(* IEC 61131-3 sources: MessageBox/src/Ar/MessageBox, 3 files *)

(* ---- MessageBox.typ ---- *)
(*
* File: MessageBox.typ
* Copyright (c) 2023 Loupe
* https://loupe.team
*
* This file is part of MessageBox, licensed under the MIT License.
*
*)
(*Popup HMI Control*)

TYPE
	MessageBox_HMI_typ : 	STRUCT
		Layer : MessageBox_Layer_typ;
		TextSnippets : MessageBox_TextSnippets;
		Prompt : HMI_TextBox_typ;
		UserInput : HMI_TextBox_typ;
		Buttons1 : HMI_Button_typ;
		Buttons2 : HMI_Button_typ;
		Buttons3 : HMI_Button_typ;
		Buttons4 : HMI_Button_typ;
		Buttons5 : HMI_Button_typ;
		Internal : MessageBox_HMI_Internal_typ;
	END_STRUCT;
END_TYPE

(*Popup HMI Mapping*)

TYPE
	MessageBox_TextSnippets : 	STRUCT
		Message : STRING[260];
		UserString : STRING[260];
		Buttons1 : STRING[80];
		Buttons2 : STRING[80];
		Buttons3 : STRING[80];
		Buttons4 : STRING[80];
		Buttons5 : STRING[80];
	END_STRUCT;
	MessageBox_Layer_typ : 	STRUCT
		Active : BOOL;
		Status : UINT;
	END_STRUCT;
END_TYPE

(*Structure to create a message*)

TYPE
	MessageBox_Message_typ : 	STRUCT
		Prompt : MessageBox_Message_Prompt_typ;
		Buttons : ARRAY[0..4]OF MessageBox_Button_typ;
		pUserString : UDINT;
		MessageID : UDINT;
	END_STRUCT;
	MessageBox_Message_Prompt_typ : 	STRUCT
		pText : UDINT;
		Index : UINT;
	END_STRUCT;
	MessageBox_Button_typ : 	STRUCT
		pText : UDINT;
		Index : UINT;
		pCmd : UDINT;
	END_STRUCT;
END_TYPE

(*Popup Backend*)

TYPE
	MessageBox_typ : 	STRUCT
		Internal : MessageBox_Internal_typ;
	END_STRUCT;
	MessageBox_Internal_typ : 	STRUCT
		Buffer : Buffer_typ;
	END_STRUCT;
	MessageBox_HMI_Internal_typ : 	STRUCT
		Message : MessageBox_Message_typ;
		_Show : BOOL;
		_CMD : ARRAY[0..4]OF BOOL;
		_ShowEdge : BOOL;
		_ShowDelay : TON;
		_MessageID : UDINT;
	END_STRUCT;
END_TYPE

(*Errors*)

TYPE
	MESSAGE_ERR :
		(
		MESSAGE_ERR_INVALID_ID,
		MESSAGE_ERR_ALREADY_INIT,
		MESSAGE_ERR_OUT_OF_MEMORY,
		MESSAGE_ERR_BUFFER_FULL,
		MESSAGE_ERR_UNINITIALIZED,
		MESSAGE_ERR_EMPTY,
		MESSAGE_ERR_INVALID_POINTER,
		MESSAGE_ERR_
		);
END_TYPE

(* ---- MessageBox.fun ---- *)
(*
* File: MessageBox.fun
* Copyright (c) 2023 Loupe
* https://loupe.team
*
* This file is part of MessageBox, licensed under the MIT License.
*
*)

FUNCTION MessageBox_Init : UDINT (*instantiates a message queue*)
	VAR_INPUT
		QueueSize : USINT;
	END_VAR
END_FUNCTION

FUNCTION MessageBox_AddMsg : UDINT (*adds a normal priority message to the bottom of the list*)
	VAR_INPUT
		Message : UDINT;
		Button1Text : UDINT;
		pCommand1 : UDINT;
		Button2Text : UDINT;
		pCommand2 : UDINT;
	END_VAR
END_FUNCTION

FUNCTION MessageBox_AddMsgTop : UDINT (*adds a high priority message to the top of the list, can bump off the last msg in the buffer*)
	VAR_INPUT
		Message : UDINT;
		Button1Text : UDINT;
		pCommand1 : UDINT;
		Button2Text : UDINT;
		pCommand2 : UDINT;
	END_VAR
END_FUNCTION

FUNCTION PromptBox_AddMsg : UDINT (*adds a normal priority message to the bottom of the list*)
	VAR_INPUT
		Message : UDINT;
		pInputString : UDINT;
		Button1Text : UDINT;
		pCommand1 : UDINT;
		Button2Text : UDINT;
		pCommand2 : UDINT;
	END_VAR
END_FUNCTION

FUNCTION PromptBox_AddMsgTop : UDINT (*adds a high priority message to the top of the list, can bump off the last msg in the buffer*)
	VAR_INPUT
		Message : UDINT;
		pInputString : UDINT;
		Button1Text : UDINT;
		pCommand1 : UDINT;
		Button2Text : UDINT;
		pCommand2 : UDINT;
	END_VAR
END_FUNCTION

FUNCTION MessageBox_RemoveMsg : UDINT (*marks a message for removal based on messageID*)
	VAR_INPUT
		MessageID : UDINT;
	END_VAR
END_FUNCTION

FUNCTION MessageBox_HMI : UDINT (*used to cyclically update messagebox interface with HMI*)
	VAR_INPUT
		MessageBox : MessageBox_HMI_typ;
	END_VAR
END_FUNCTION

FUNCTION MessageBox_Add3BtnMsg : UDINT (*adds a normal priority 3-button message to the bottom of the list*)
	VAR_INPUT
		Message : UDINT;
		Button1Text : UDINT;
		pCommand1 : UDINT;
		Button2Text : UDINT;
		pCommand2 : UDINT;
		Button3Text : UDINT;
		pCommand3 : UDINT;
	END_VAR
END_FUNCTION

FUNCTION MessageBox_Add3BtnMsgTop : UDINT (*adds a high priority 3-button message to the top of the list, can bump off the last msg in the buffer*)
	VAR_INPUT
		Message : UDINT;
		Button1Text : UDINT;
		pCommand1 : UDINT;
		Button2Text : UDINT;
		pCommand2 : UDINT;
		Button3Text : UDINT;
		pCommand3 : UDINT;
	END_VAR
END_FUNCTION

FUNCTION PromptBox_Add3BtnMsg : UDINT (*adds a normal priority 3-button message to the bottom of the list*)
	VAR_INPUT
		Message : UDINT;
		pInputString : UDINT;
		Button1Text : UDINT;
		pCommand1 : UDINT;
		Button2Text : UDINT;
		pCommand2 : UDINT;
		Button3Text : UDINT;
		pCommand3 : UDINT;
	END_VAR
END_FUNCTION

FUNCTION PromptBox_Add3BtnMsgTop : UDINT (*adds a high priority 3-button message to the top of the list, can bump off the last msg in the buffer*)
	VAR_INPUT
		Message : UDINT;
		pInputString : UDINT;
		Button1Text : UDINT;
		pCommand1 : UDINT;
		Button2Text : UDINT;
		pCommand2 : UDINT;
		Button3Text : UDINT;
		pCommand3 : UDINT;
	END_VAR
END_FUNCTION

FUNCTION MessageBox_AddNBtnMsg : UDINT (*adds a normal priority N-button message (N <= 5) to the bottom of the list*)
	VAR_INPUT
		Message : UDINT;
		Button1Text : UDINT;
		pCommand1 : UDINT;
		Button2Text : UDINT;
		pCommand2 : UDINT;
		Button3Text : UDINT;
		pCommand3 : UDINT;
		Button4Text : UDINT;
		pCommand4 : UDINT;
		Button5Text : UDINT;
		pCommand5 : UDINT;
	END_VAR
END_FUNCTION

FUNCTION MessageBox_AddNBtnMsgTop : UDINT (*adds a high priority N-button message (N <= 5) to the top of the list, can bump off the last msg in the buffer*)
	VAR_INPUT
		Message : UDINT;
		Button1Text : UDINT;
		pCommand1 : UDINT;
		Button2Text : UDINT;
		pCommand2 : UDINT;
		Button3Text : UDINT;
		pCommand3 : UDINT;
		Button4Text : UDINT;
		pCommand4 : UDINT;
		Button5Text : UDINT;
		pCommand5 : UDINT;
	END_VAR
END_FUNCTION

FUNCTION PromptBox_AddNBtnMsg : UDINT (*adds a normal priority N-button message (N <= 5) to the bottom of the list*)
	VAR_INPUT
		Message : UDINT;
		pInputString : UDINT;
		Button1Text : UDINT;
		pCommand1 : UDINT;
		Button2Text : UDINT;
		pCommand2 : UDINT;
		Button3Text : UDINT;
		pCommand3 : UDINT;
		Button4Text : UDINT;
		pCommand4 : UDINT;
		Button5Text : UDINT;
		pCommand5 : UDINT;
	END_VAR
END_FUNCTION

FUNCTION PromptBox_AddNBtnMsgTop : UDINT (*adds a high priority N-button message (N <= 5) to the top of the list, can bump off the last msg in the buffer*)
	VAR_INPUT
		Message : UDINT;
		pInputString : UDINT;
		Button1Text : UDINT;
		pCommand1 : UDINT;
		Button2Text : UDINT;
		pCommand2 : UDINT;
		Button3Text : UDINT;
		pCommand3 : UDINT;
		Button4Text : UDINT;
		pCommand4 : UDINT;
		Button5Text : UDINT;
		pCommand5 : UDINT;
	END_VAR
END_FUNCTION

(* ---- MessageBox.var ---- *)
(*
* File: MessageBox.var
* Copyright (c) 2023 Loupe
* https://loupe.team
*
* This file is part of MessageBox, licensed under the MIT License.
*
*)
VAR CONSTANT
	MESSAGEBOX_MAX : UINT := 5;
	MESSAGEBOX_MESSAGE_LENGTH : UINT := 80;
END_VAR
